FUNCTION_BLOCK FB_HMI_SERVICES EXTENDS FB_HMI_COMPONENT
VAR_INPUT
END_VAR
VAR_OUTPUT
END_VAR
VAR_IN_OUT
    fbInstance : FB_SERVICES;
END_VAR
VAR
    fbTime : FB_HMI_SERVICES_TIME;
END_VAR

fbTime(fbInstance := fbInstance.fbTime);

fbHealthStatus(
    bIsEnabled  := fbTime.fbHealthStatus.bEnabled,
    bIsGood     := fbTime.fbHealthStatus.bGood);
fbBusyStatus(
    bIsEnabled  := fbTime.fbBusyStatus.bEnabled,
    bIsBusy     := fbTime.fbBusyStatus.bBusy);

M_UpdateStatusColor();

END_FUNCTION_BLOCK

(* stored: Version 1.1.0.1, ProductVersion 3.1.4024.14
   POU FB_HMI_SERVICES: Id {d0e78a0c-6b15-4173-ac07-9bdbb6997828}, SpecialFunc None *)
